FUNCTION_BLOCK PUBL_0 (* Event-only Local Publisher *)
  (* Standard: 61499-1; Classification: Communications; Description: Local multicast group publisher *)
  (* Version 0.0, 2002-05-02, JHC, Rockwell Automation, Optimized version. *)
  (* Version 0.0, 2001-10-02, JHC, Rockwell Automation, Copied/Modified from PUBLISH *)
  (* Compiler header: package fb.rt.net; *)
  (* Compiler Java IBM VisualAge 3.0 *)
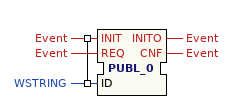
  EVENT_INPUT
    INIT WITH ID; (* Service Initialization *)
    REQ; (* Service Request *)
  END_EVENT
  EVENT_OUTPUT
    INITO; (* Initialization Confirm *)
    CNF; (* Service Confirmation *)
  END_EVENT
  VAR_INPUT
    ID : WSTRING; (* Local Group Name-Default is FB Instance Name *)
  END_VAR
  SERVICE PUBL_0/SUBL_0 (* Event Publication Service *)
    SEQUENCE normal_establishment
      PUBL_0.INIT(ID) -> PUBL_0.INITO();
      SUBL_0.INIT(ID) -> SUBL_0.INITO();
    END_SEQUENCE
    SEQUENCE event_transfer
      PUBL_0.REQ() -> SUBL_0.IND() -> PUBL_0.CNF();
    END_SEQUENCE
  END_SERVICE
END_FUNCTION_BLOCK
